(* Logix 5000 project; controller Week_3_PLC_1_Traffic_Light_Ver_2 Emulate 5570 rev 30.12; software revision 30.01 *)

TASK MainTask (continuous, watchdog 500 ms) : MainProgram

MODULES
   Local : Emulate 5570 (ICP 2, rev 30.12)
END_MODULES

PROGRAM MainProgram   (* main routine MainRoutine *)
VAR
   NS_GREEN : BOOL;
   NS_RED : BOOL;
   NS_YELLOW : BOOL;
   Power : BOOL;
   Start : BOOL;
   Stop : BOOL;
   Timer : TIMER := (PRE := 28000);
   WE_GREEN : BOOL;
   WE_RED : BOOL;
   WE_YELLOW : BOOL;
END_VAR

ROUTINE MainRoutine   (* ladder *)
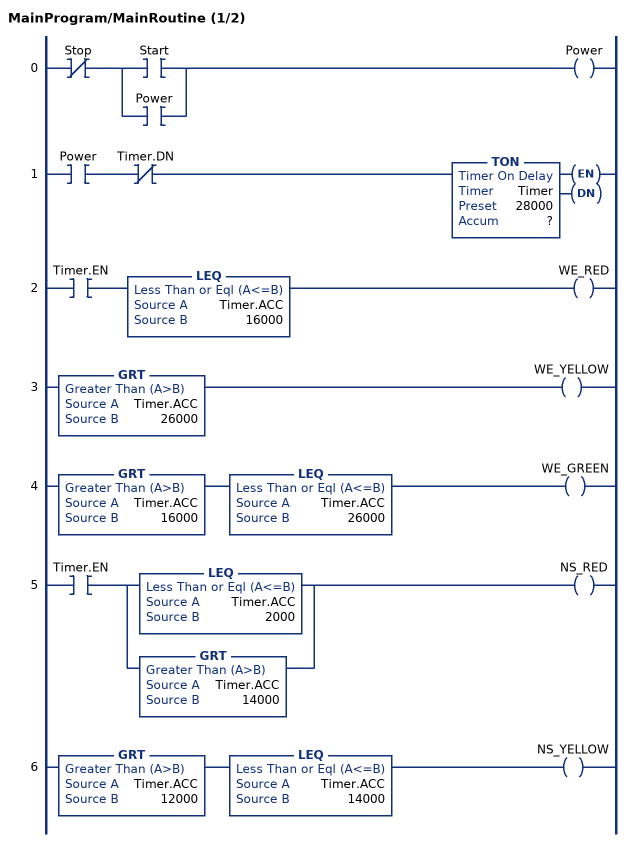
   0: XIO(Stop)[XIC(Start) ,XIC(Power) ]OTE(Power);
   1: XIC(Power)XIO(Timer.DN)TON(Timer,?,?);
   2: XIC(Timer.EN)LEQ(Timer.ACC,16000)OTE(WE_RED);
   3: GRT(Timer.ACC,26000)OTE(WE_YELLOW);
   4: GRT(Timer.ACC,16000)LEQ(Timer.ACC,26000)OTE(WE_GREEN);
   5: XIC(Timer.EN)[LEQ(Timer.ACC,2000) ,GRT(Timer.ACC,14000) ]OTE(NS_RED);
   6: GRT(Timer.ACC,12000)LEQ(Timer.ACC,14000)OTE(NS_YELLOW);
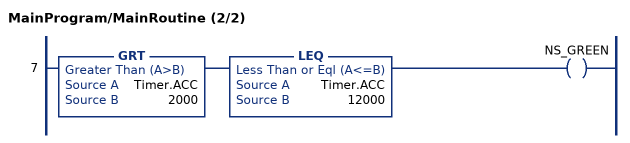
   7: GRT(Timer.ACC,2000)LEQ(Timer.ACC,12000)OTE(NS_GREEN);
END_ROUTINE
END_PROGRAM
